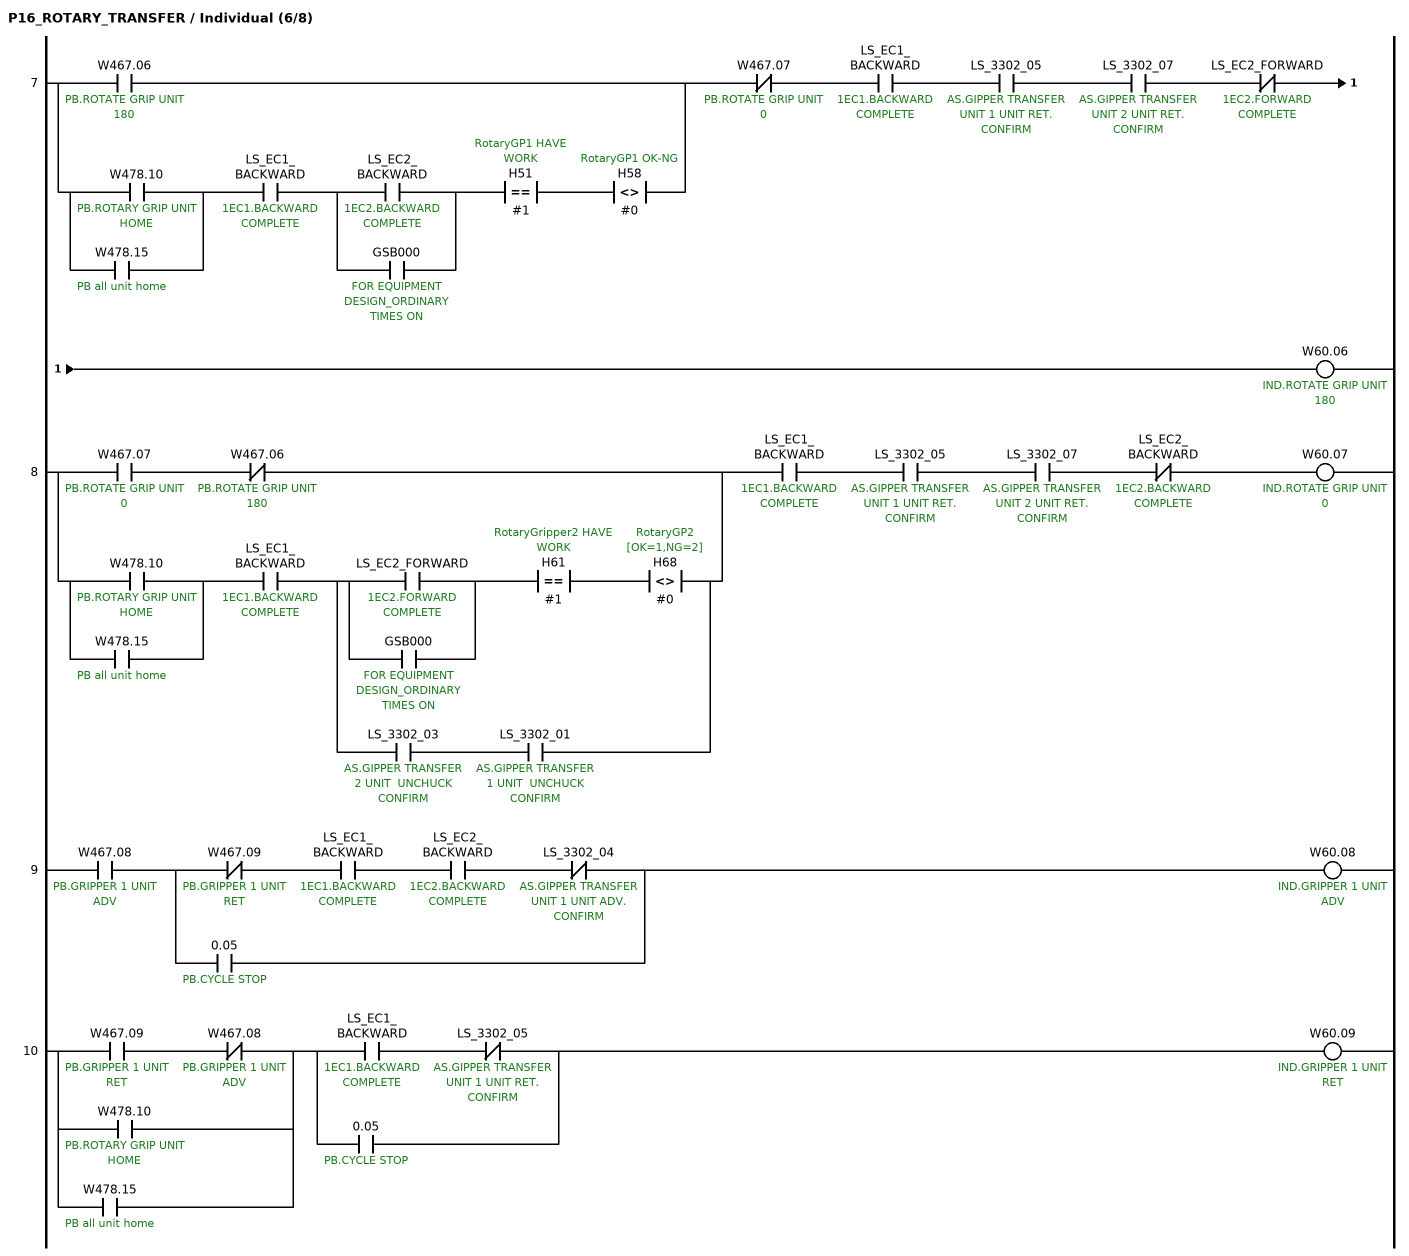
; [picture p288: P16_ROTARY_TRANSFER / Individual, rungs 7-10]
; rung 7
LD W467.06  ; PB.ROTATE GRIP UNIT 180
LD W478.10  ; PB.ROTARY GRIP UNIT HOME
OR W478.15  ; PB all unit home
AND LS_EC1_BACKWARD  ; 1EC1.BACKWARD COMPLETE
LD LS_EC2_BACKWARD  ; 1EC2.BACKWARD COMPLETE
OR GSB000  ; FOR EQUIPMENT DESIGN_ORDINARY TIMES ON
ANDLD
AND=(300) H51 #1  ; RotaryGP1 HAVE WORK
AND<>(305) H58 #0  ; RotaryGP1 OK-NG
ORLD
ANDNOT W467.07  ; PB.ROTATE GRIP UNIT 0
AND LS_EC1_BACKWARD  ; 1EC1.BACKWARD COMPLETE
AND LS_3302_05  ; AS.GIPPER TRANSFER UNIT 1 UNIT RET. CONFIRM
AND LS_3302_07  ; AS.GIPPER TRANSFER UNIT 2 UNIT RET. CONFIRM
ANDNOT LS_EC2_FORWARD  ; 1EC2.FORWARD COMPLETE
OUT W60.06  ; IND.ROTATE GRIP UNIT 180
; rung 8
LD W467.07  ; PB.ROTATE GRIP UNIT 0
ANDNOT W467.06  ; PB.ROTATE GRIP UNIT 180
LD W478.10  ; PB.ROTARY GRIP UNIT HOME
OR W478.15  ; PB all unit home
AND LS_EC1_BACKWARD  ; 1EC1.BACKWARD COMPLETE
LD LS_EC2_FORWARD  ; 1EC2.FORWARD COMPLETE
OR GSB000  ; FOR EQUIPMENT DESIGN_ORDINARY TIMES ON
AND=(300) H61 #1  ; RotaryGripper2 HAVE WORK
AND<>(305) H68 #0  ; RotaryGP2 [OK=1,NG=2]
LD LS_3302_03  ; AS.GIPPER TRANSFER 2 UNIT  UNCHUCK CONFIRM
AND LS_3302_01  ; AS.GIPPER TRANSFER 1 UNIT  UNCHUCK CONFIRM
ORLD
ANDLD
ORLD
AND LS_EC1_BACKWARD  ; 1EC1.BACKWARD COMPLETE
AND LS_3302_05  ; AS.GIPPER TRANSFER UNIT 1 UNIT RET. CONFIRM
AND LS_3302_07  ; AS.GIPPER TRANSFER UNIT 2 UNIT RET. CONFIRM
ANDNOT LS_EC2_BACKWARD  ; 1EC2.BACKWARD COMPLETE
OUT W60.07  ; IND.ROTATE GRIP UNIT 0
; rung 9
LD W467.08  ; PB.GRIPPER 1 UNIT ADV
LDNOT W467.09  ; PB.GRIPPER 1 UNIT RET
AND LS_EC1_BACKWARD  ; 1EC1.BACKWARD COMPLETE
AND LS_EC2_BACKWARD  ; 1EC2.BACKWARD COMPLETE
ANDNOT LS_3302_04  ; AS.GIPPER TRANSFER UNIT 1 UNIT ADV. CONFIRM
OR 0.05  ; PB.CYCLE STOP
ANDLD
OUT W60.08  ; IND.GRIPPER 1 UNIT ADV
; rung 10
LD W467.09  ; PB.GRIPPER 1 UNIT RET
ANDNOT W467.08  ; PB.GRIPPER 1 UNIT ADV
OR W478.10  ; PB.ROTARY GRIP UNIT HOME
OR W478.15  ; PB all unit home
LD LS_EC1_BACKWARD  ; 1EC1.BACKWARD COMPLETE
ANDNOT LS_3302_05  ; AS.GIPPER TRANSFER UNIT 1 UNIT RET. CONFIRM
OR 0.05  ; PB.CYCLE STOP
ANDLD
OUT W60.09  ; IND.GRIPPER 1 UNIT RET

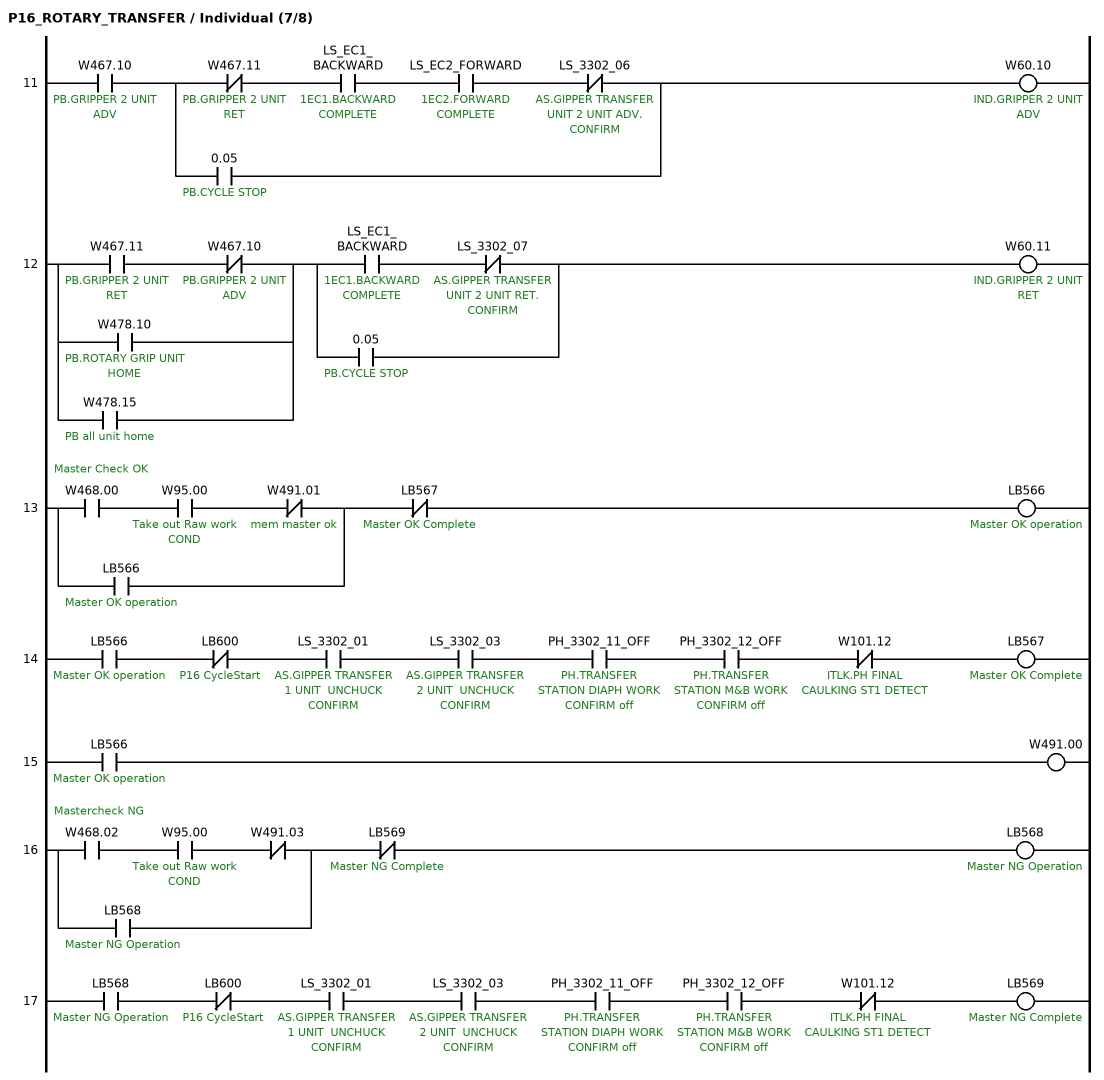
; rung 11
LD W467.10  ; PB.GRIPPER 2 UNIT ADV
LDNOT W467.11  ; PB.GRIPPER 2 UNIT RET
AND LS_EC1_BACKWARD  ; 1EC1.BACKWARD COMPLETE
AND LS_EC2_FORWARD  ; 1EC2.FORWARD COMPLETE
ANDNOT LS_3302_06  ; AS.GIPPER TRANSFER UNIT 2 UNIT ADV. CONFIRM
OR 0.05  ; PB.CYCLE STOP
ANDLD
OUT W60.10  ; IND.GRIPPER 2 UNIT ADV
; rung 12
LD W467.11  ; PB.GRIPPER 2 UNIT RET
ANDNOT W467.10  ; PB.GRIPPER 2 UNIT ADV
OR W478.10  ; PB.ROTARY GRIP UNIT HOME
OR W478.15  ; PB all unit home
LD LS_EC1_BACKWARD  ; 1EC1.BACKWARD COMPLETE
ANDNOT LS_3302_07  ; AS.GIPPER TRANSFER UNIT 2 UNIT RET. CONFIRM
OR 0.05  ; PB.CYCLE STOP
ANDLD
OUT W60.11  ; IND.GRIPPER 2 UNIT RET
; rung 13: Master Check OK
LD W468.00
AND W95.00  ; Take out Raw work COND
ANDNOT W491.01  ; mem master ok
OR LB566  ; Master OK operation
ANDNOT LB567  ; Master OK Complete
OUT LB566  ; Master OK operation
; rung 14
LD LB566  ; Master OK operation
ANDNOT LB600  ; P16 CycleStart
AND LS_3302_01  ; AS.GIPPER TRANSFER 1 UNIT  UNCHUCK CONFIRM
AND LS_3302_03  ; AS.GIPPER TRANSFER 2 UNIT  UNCHUCK CONFIRM
AND PH_3302_11_OFF  ; PH.TRANSFER STATION DIAPH WORK CONFIRM off
AND PH_3302_12_OFF  ; PH.TRANSFER STATION M&B WORK CONFIRM off
ANDNOT W101.12  ; ITLK.PH FINAL CAULKING ST1 DETECT
OUT LB567  ; Master OK Complete
; rung 15
LD LB566  ; Master OK operation
OUT W491.00
; rung 16: Mastercheck NG
LD W468.02
AND W95.00  ; Take out Raw work COND
ANDNOT W491.03
OR LB568  ; Master NG Operation
ANDNOT LB569  ; Master NG Complete
OUT LB568  ; Master NG Operation
; rung 17
LD LB568  ; Master NG Operation
ANDNOT LB600  ; P16 CycleStart
AND LS_3302_01  ; AS.GIPPER TRANSFER 1 UNIT  UNCHUCK CONFIRM
AND LS_3302_03  ; AS.GIPPER TRANSFER 2 UNIT  UNCHUCK CONFIRM
AND PH_3302_11_OFF  ; PH.TRANSFER STATION DIAPH WORK CONFIRM off
AND PH_3302_12_OFF  ; PH.TRANSFER STATION M&B WORK CONFIRM off
ANDNOT W101.12  ; ITLK.PH FINAL CAULKING ST1 DETECT
OUT LB569  ; Master NG Complete

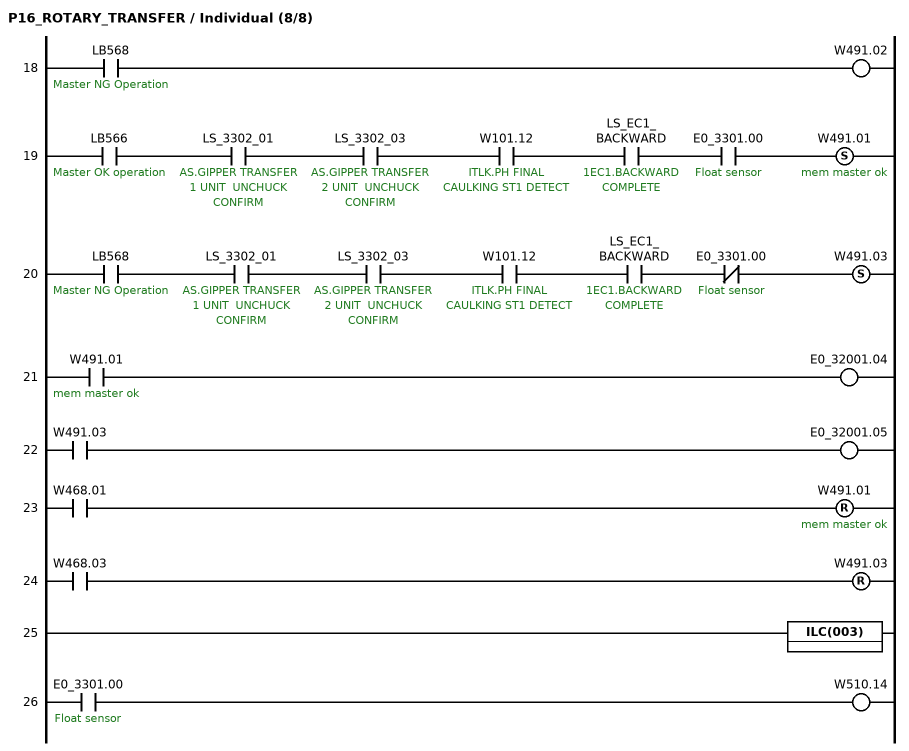
; rung 18
LD LB568  ; Master NG Operation
OUT W491.02
; rung 19
LD LB566  ; Master OK operation
AND LS_3302_01  ; AS.GIPPER TRANSFER 1 UNIT  UNCHUCK CONFIRM
AND LS_3302_03  ; AS.GIPPER TRANSFER 2 UNIT  UNCHUCK CONFIRM
AND W101.12  ; ITLK.PH FINAL CAULKING ST1 DETECT
AND LS_EC1_BACKWARD  ; 1EC1.BACKWARD COMPLETE
AND E0_3301.00  ; Float sensor
SET W491.01  ; mem master ok
; rung 20
LD LB568  ; Master NG Operation
AND LS_3302_01  ; AS.GIPPER TRANSFER 1 UNIT  UNCHUCK CONFIRM
AND LS_3302_03  ; AS.GIPPER TRANSFER 2 UNIT  UNCHUCK CONFIRM
AND W101.12  ; ITLK.PH FINAL CAULKING ST1 DETECT
AND LS_EC1_BACKWARD  ; 1EC1.BACKWARD COMPLETE
ANDNOT E0_3301.00  ; Float sensor
SET W491.03
; rung 21
LD W491.01  ; mem master ok
OUT E0_32001.04
; rung 22
LD W491.03
OUT E0_32001.05
; rung 23
LD W468.01
RSET W491.01  ; mem master ok
; rung 24
LD W468.03
RSET W491.03
; rung 25
ILC(003)
; rung 26
LD E0_3301.00  ; Float sensor
OUT W510.14

### Section END
; rung 0
END(001)

## Program P17_OK_NG_DISCHARGE (cyclic task 7)
Local symbols
LB2199 E0_46.15 BOOL  ; P16 AutoCycleEnd
LB2200 E0_41.02 BOOL  ; AUTO START BEGIN
LB2201 E0_41.03 BOOL  ; SOL.WORK FINISH TRAY DOWN
LB2202 E0_41.04 BOOL  ; SOL.WORK FINISH TRAY DOWN CONF
LB2203 E0_41.05 BOOL  ; SOL.OK PUSH UP
LB2204 E0_41.06 BOOL  ; SOL.OK PUSH UP CONF
LB2205 E0_41.07 BOOL  ; OK DISCHARGE CONFIRM
LB2206 E0_41.08 BOOL  ; SOL.OK PUSH DOWN
LB2207 E0_41.09 BOOL  ; SOL.OK PUSH DOWN CONF
LB2208 E0_41.10 BOOL  ; SOL.WORK FINISH TRAY UP
LB2209 E0_41.11 BOOL  ; SOL.WORK FINISH TRAY UP CONF
LB2210 E0_41.12 BOOL  ; AUTO START BEGIN
LB2211 E0_41.13 BOOL  ; SOL.WORK FINISH TRAY DOWN
LB2212 E0_41.14 BOOL  ; SOL.WORK FINISH TRAY DOWN CONF
LB2213 E0_41.15 BOOL  ; SOL.NG PUSH DOWN
LB2214 E0_42.00 BOOL  ; SOL.NG PUSH DOWN CONF
LB2215 E0_42.01 BOOL  ; NG DISCHARGE CONFIRM
LB2216 E0_42.02 BOOL  ; SOL.NG PUSH UP
LB2217 E0_42.03 BOOL  ; SOL.NG PUSH UP CONF
LB2218 E0_42.04 BOOL  ; SOL.WORK FINISH TRAY UP
LB2219 E0_42.05 BOOL  ; SOL.WORK FINISH TRAY UP CONF
LB2397 E0_42.06 BOOL  ; P16 OK Discharge END
LB2398 E0_42.07 BOOL  ; P16 NG Discharge END
LB2399 E0_42.08 BOOL  ; P17 AutoCycleEnd
LB432 E0_47.00 BOOL  ; IND 1 CYCLE
LB700 E0_42.09 BOOL  ; P17 CycleStart
LB701 E0_42.10 BOOL  ; P17 OK Discharge
LB702 E0_42.11 BOOL  ; P17 NG Discharge
LT2214 T3020 TIMER
LT231 T3024 TIMER
LT232 T3028 TIMER
trial_cv E0_46.02 BOOL

### Section Autorun

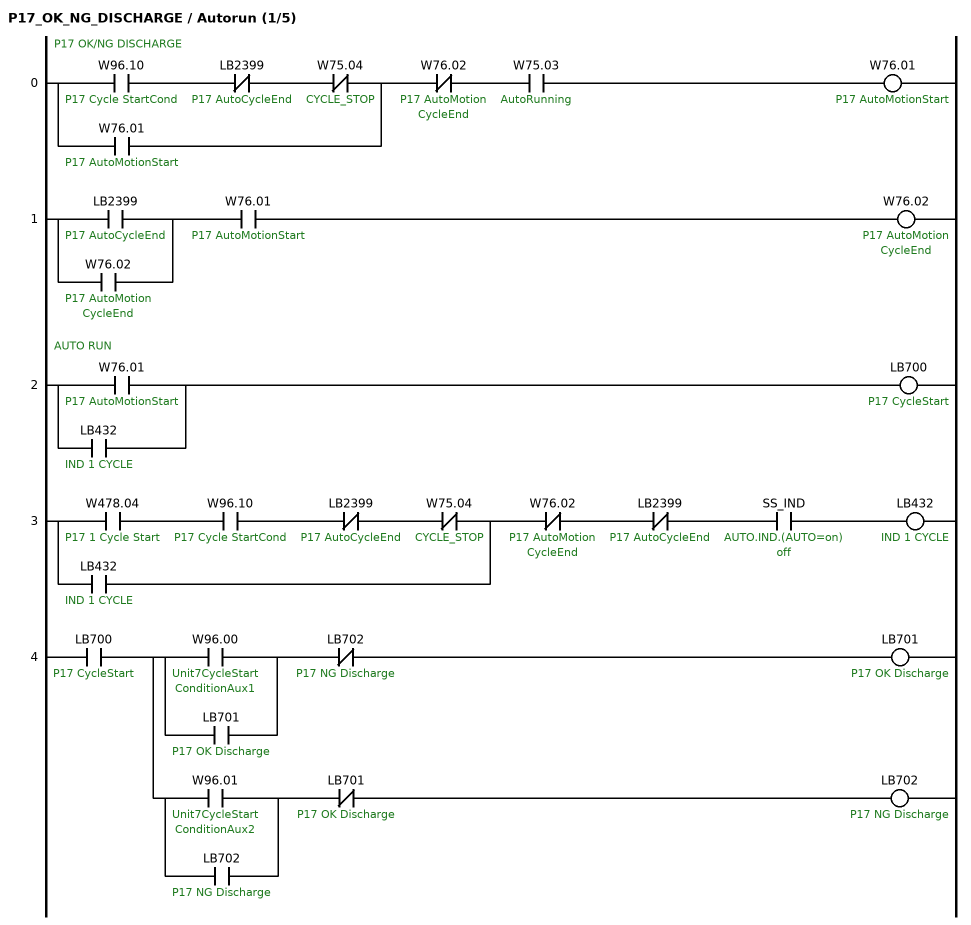
; rung 0: P17 OK/NG DISCHARGE
LD W96.10  ; P17 Cycle StartCond
ANDNOT LB2399  ; P17 AutoCycleEnd
ANDNOT W75.04  ; CYCLE_STOP
OR W76.01  ; P17 AutoMotionStart
ANDNOT W76.02  ; P17 AutoMotion CycleEnd
AND W75.03  ; AutoRunning
OUT W76.01  ; P17 AutoMotionStart
; rung 1
LD LB2399  ; P17 AutoCycleEnd
OR W76.02  ; P17 AutoMotion CycleEnd
AND W76.01  ; P17 AutoMotionStart
OUT W76.02  ; P17 AutoMotion CycleEnd
; rung 2: AUTO RUN
LD W76.01  ; P17 AutoMotionStart
OR LB432  ; IND 1 CYCLE
OUT LB700  ; P17 CycleStart
; rung 3
LD W478.04  ; P17 1 Cycle Start
AND W96.10  ; P17 Cycle StartCond
ANDNOT LB2399  ; P17 AutoCycleEnd
ANDNOT W75.04  ; CYCLE_STOP
OR LB432  ; IND 1 CYCLE
ANDNOT W76.02  ; P17 AutoMotion CycleEnd
ANDNOT LB2399  ; P17 AutoCycleEnd
AND SS_IND  ; AUTO.IND.(AUTO=on) off
OUT LB432  ; IND 1 CYCLE
; rung 4
LD LB700  ; P17 CycleStart
OUT TR0
LD W96.00  ; Unit7CycleStartConditionAux1
OR LB701  ; P17 OK Discharge
ANDLD
ANDNOT LB702  ; P17 NG Discharge
OUT LB701  ; P17 OK Discharge
LD TR0
LD W96.01  ; Unit7CycleStartConditionAux2
OR LB702  ; P17 NG Discharge
ANDLD
ANDNOT LB701  ; P17 OK Discharge
OUT LB702  ; P17 NG Discharge

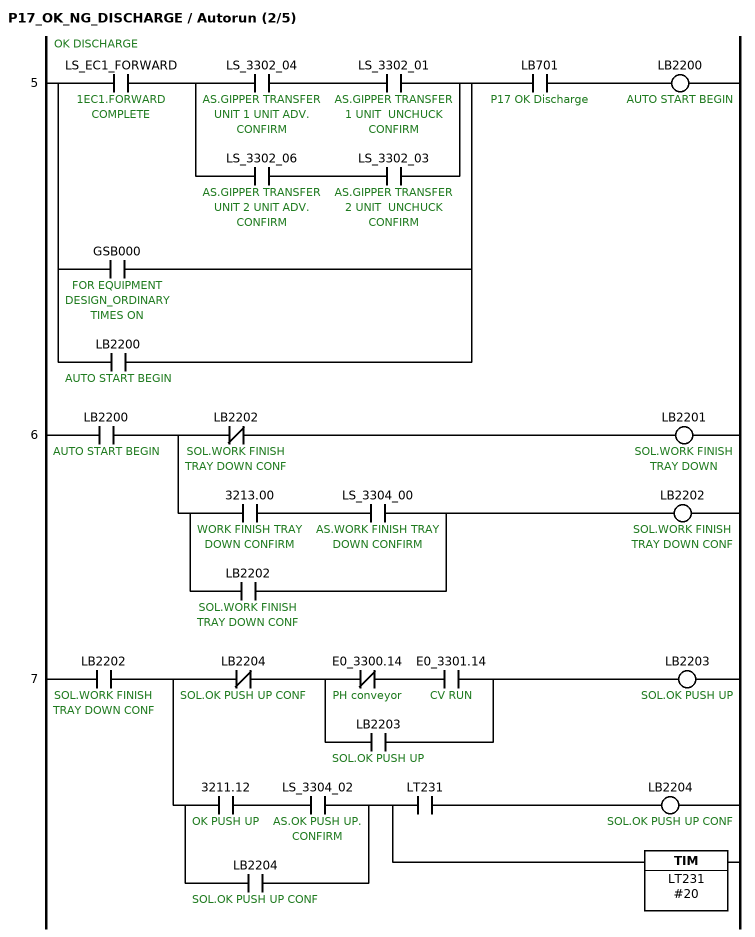
; rung 5: OK DISCHARGE
LD LS_EC1_FORWARD  ; 1EC1.FORWARD COMPLETE
LD LS_3302_04  ; AS.GIPPER TRANSFER UNIT 1 UNIT ADV. CONFIRM
AND LS_3302_01  ; AS.GIPPER TRANSFER 1 UNIT  UNCHUCK CONFIRM
LD LS_3302_06  ; AS.GIPPER TRANSFER UNIT 2 UNIT ADV. CONFIRM
AND LS_3302_03  ; AS.GIPPER TRANSFER 2 UNIT  UNCHUCK CONFIRM
ORLD
ANDLD
OR GSB000  ; FOR EQUIPMENT DESIGN_ORDINARY TIMES ON
OR LB2200  ; AUTO START BEGIN
AND LB701  ; P17 OK Discharge
OUT LB2200  ; AUTO START BEGIN
; rung 6
LD LB2200  ; AUTO START BEGIN
OUT TR0
ANDNOT LB2202  ; SOL.WORK FINISH TRAY DOWN CONF
OUT LB2201  ; SOL.WORK FINISH TRAY DOWN
LD TR0
LD 3213.00  ; WORK FINISH TRAY DOWN CONFIRM
AND LS_3304_00  ; AS.WORK FINISH TRAY DOWN CONFIRM
OR LB2202  ; SOL.WORK FINISH TRAY DOWN CONF
ANDLD
OUT LB2202  ; SOL.WORK FINISH TRAY DOWN CONF
; rung 7
LD LB2202  ; SOL.WORK FINISH TRAY DOWN CONF
OUT TR0
ANDNOT LB2204  ; SOL.OK PUSH UP CONF
LDNOT E0_3300.14  ; PH conveyor
AND E0_3301.14  ; CV RUN
OR LB2203  ; SOL.OK PUSH UP
ANDLD
OUT LB2203  ; SOL.OK PUSH UP
LD TR0
LD 3211.12  ; OK PUSH UP
AND LS_3304_02  ; AS.OK PUSH UP. CONFIRM
OR LB2204  ; SOL.OK PUSH UP CONF
ANDLD
OUT TR0
AND LT231
OUT LB2204  ; SOL.OK PUSH UP CONF
LD TR0
TIM LT231 #20

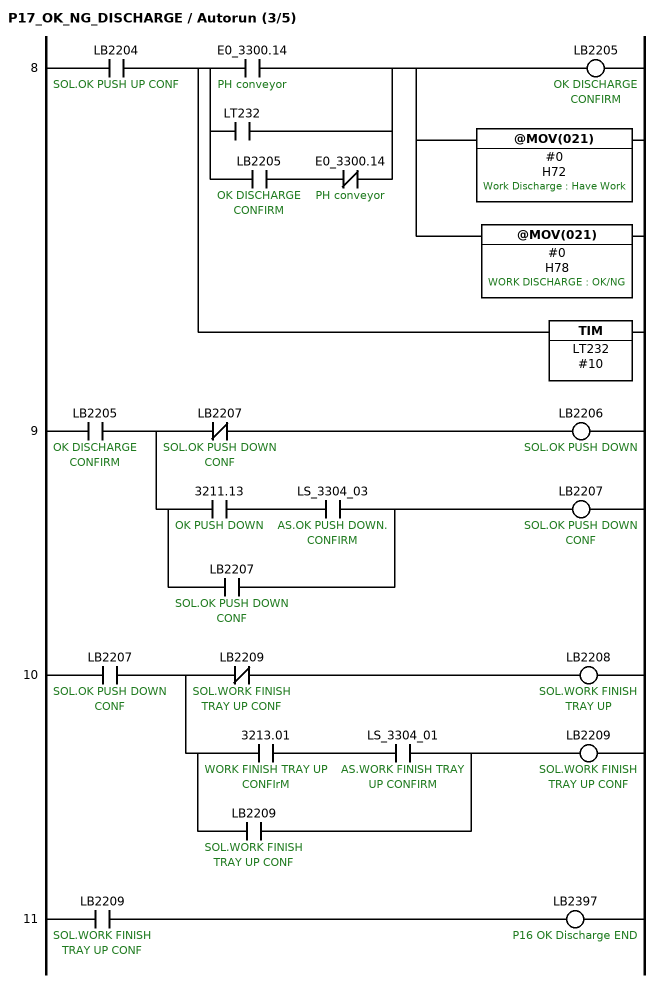
; rung 8
LD LB2204  ; SOL.OK PUSH UP CONF
OUT TR0
LD E0_3300.14  ; PH conveyor
OR LT232
LD LB2205  ; OK DISCHARGE CONFIRM
ANDNOT E0_3300.14  ; PH conveyor
ORLD
ANDLD
OUT LB2205  ; OK DISCHARGE CONFIRM
@MOV(021) #0 H72  ; Work Discharge : Have Work
@MOV(021) #0 H78  ; WORK DISCHARGE : OK/NG
LD TR0
TIM LT232 #10
; rung 9
LD LB2205  ; OK DISCHARGE CONFIRM
OUT TR0
ANDNOT LB2207  ; SOL.OK PUSH DOWN CONF
OUT LB2206  ; SOL.OK PUSH DOWN
LD TR0
LD 3211.13  ; OK PUSH DOWN
AND LS_3304_03  ; AS.OK PUSH DOWN. CONFIRM
OR LB2207  ; SOL.OK PUSH DOWN CONF
ANDLD
OUT LB2207  ; SOL.OK PUSH DOWN CONF
; rung 10
LD LB2207  ; SOL.OK PUSH DOWN CONF
OUT TR0
ANDNOT LB2209  ; SOL.WORK FINISH TRAY UP CONF
OUT LB2208  ; SOL.WORK FINISH TRAY UP
LD TR0
LD 3213.01  ; WORK FINISH TRAY UP CONFIrM
AND LS_3304_01  ; AS.WORK FINISH TRAY UP CONFIRM
OR LB2209  ; SOL.WORK FINISH TRAY UP CONF
ANDLD
OUT LB2209  ; SOL.WORK FINISH TRAY UP CONF
; rung 11
LD LB2209  ; SOL.WORK FINISH TRAY UP CONF
OUT LB2397  ; P16 OK Discharge END

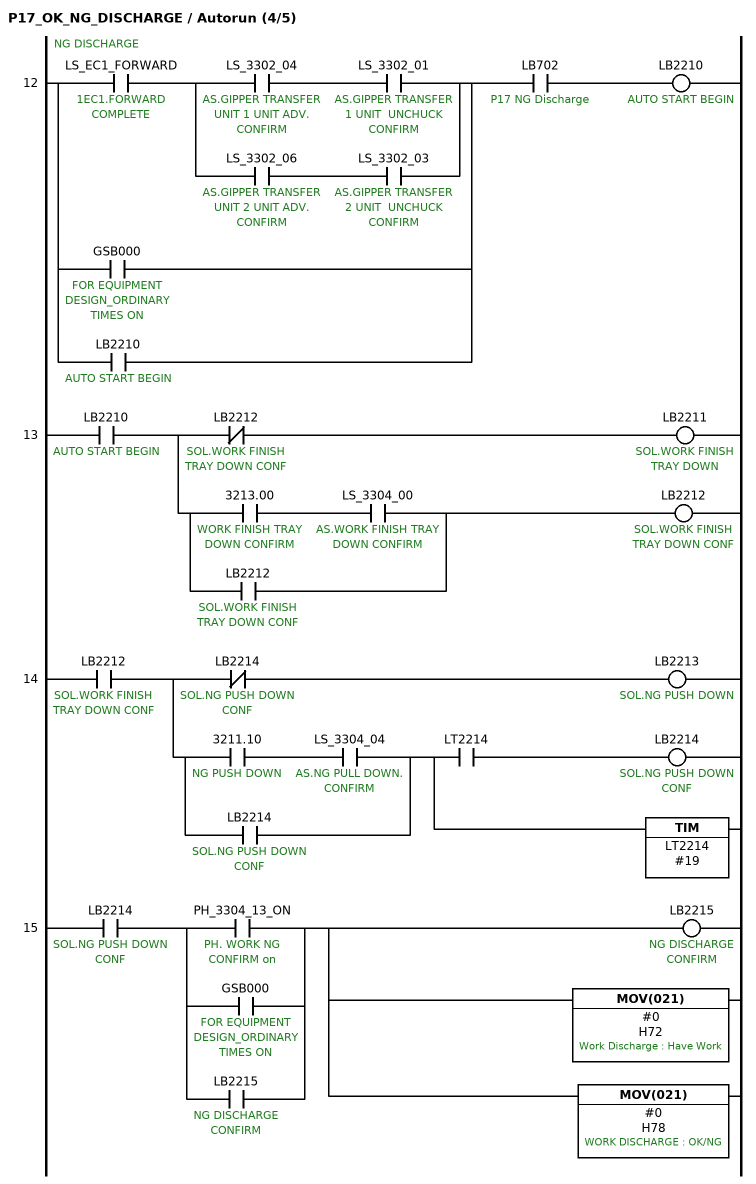
; rung 12: NG DISCHARGE
LD LS_EC1_FORWARD  ; 1EC1.FORWARD COMPLETE
LD LS_3302_04  ; AS.GIPPER TRANSFER UNIT 1 UNIT ADV. CONFIRM
AND LS_3302_01  ; AS.GIPPER TRANSFER 1 UNIT  UNCHUCK CONFIRM
LD LS_3302_06  ; AS.GIPPER TRANSFER UNIT 2 UNIT ADV. CONFIRM
AND LS_3302_03  ; AS.GIPPER TRANSFER 2 UNIT  UNCHUCK CONFIRM
ORLD
ANDLD
OR GSB000  ; FOR EQUIPMENT DESIGN_ORDINARY TIMES ON
OR LB2210  ; AUTO START BEGIN
AND LB702  ; P17 NG Discharge
OUT LB2210  ; AUTO START BEGIN
; rung 13
LD LB2210  ; AUTO START BEGIN
OUT TR0
ANDNOT LB2212  ; SOL.WORK FINISH TRAY DOWN CONF
OUT LB2211  ; SOL.WORK FINISH TRAY DOWN
LD TR0
LD 3213.00  ; WORK FINISH TRAY DOWN CONFIRM
AND LS_3304_00  ; AS.WORK FINISH TRAY DOWN CONFIRM
OR LB2212  ; SOL.WORK FINISH TRAY DOWN CONF
ANDLD
OUT LB2212  ; SOL.WORK FINISH TRAY DOWN CONF
; rung 14
LD LB2212  ; SOL.WORK FINISH TRAY DOWN CONF
OUT TR0
ANDNOT LB2214  ; SOL.NG PUSH DOWN CONF
OUT LB2213  ; SOL.NG PUSH DOWN
LD TR0
LD 3211.10  ; NG PUSH DOWN
AND LS_3304_04  ; AS.NG PULL DOWN. CONFIRM
OR LB2214  ; SOL.NG PUSH DOWN CONF
ANDLD
OUT TR0
AND LT2214
OUT LB2214  ; SOL.NG PUSH DOWN CONF
LD TR0
TIM LT2214 #19
; rung 15
LD LB2214  ; SOL.NG PUSH DOWN CONF
LD PH_3304_13_ON  ; PH. WORK NG CONFIRM on
OR GSB000  ; FOR EQUIPMENT DESIGN_ORDINARY TIMES ON
OR LB2215  ; NG DISCHARGE CONFIRM
ANDLD
OUT LB2215  ; NG DISCHARGE CONFIRM
MOV(021) #0 H72  ; Work Discharge : Have Work
MOV(021) #0 H78  ; WORK DISCHARGE : OK/NG

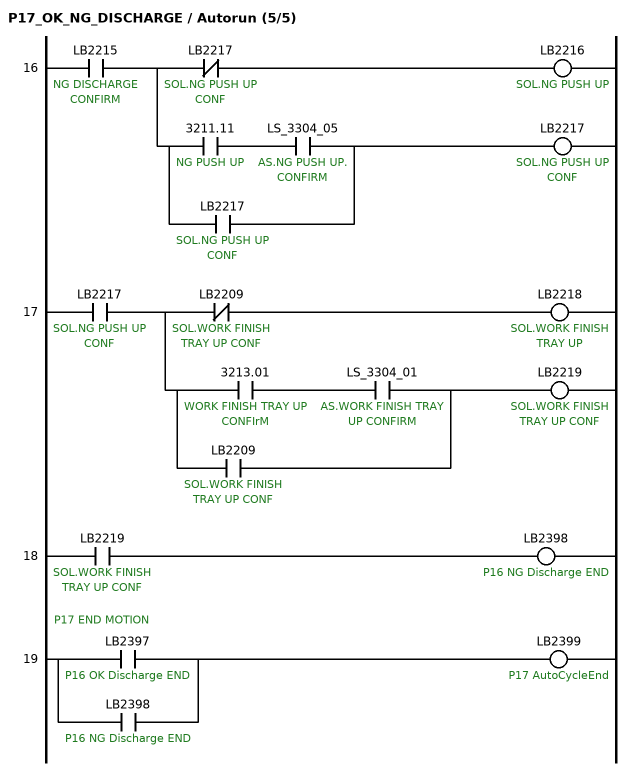
; rung 16
LD LB2215  ; NG DISCHARGE CONFIRM
OUT TR0
ANDNOT LB2217  ; SOL.NG PUSH UP CONF
OUT LB2216  ; SOL.NG PUSH UP
LD TR0
LD 3211.11  ; NG PUSH UP
AND LS_3304_05  ; AS.NG PUSH UP. CONFIRM
OR LB2217  ; SOL.NG PUSH UP CONF
ANDLD
OUT LB2217  ; SOL.NG PUSH UP CONF
; rung 17
LD LB2217  ; SOL.NG PUSH UP CONF
OUT TR0
ANDNOT LB2209  ; SOL.WORK FINISH TRAY UP CONF
OUT LB2218  ; SOL.WORK FINISH TRAY UP
LD TR0
LD 3213.01  ; WORK FINISH TRAY UP CONFIrM
AND LS_3304_01  ; AS.WORK FINISH TRAY UP CONFIRM
OR LB2209  ; SOL.WORK FINISH TRAY UP CONF
ANDLD
OUT LB2219  ; SOL.WORK FINISH TRAY UP CONF
; rung 18
LD LB2219  ; SOL.WORK FINISH TRAY UP CONF
OUT LB2398  ; P16 NG Discharge END
; rung 19: P17 END MOTION
LD LB2397  ; P16 OK Discharge END
OR LB2398  ; P16 NG Discharge END
OUT LB2399  ; P17 AutoCycleEnd

### Section Condition

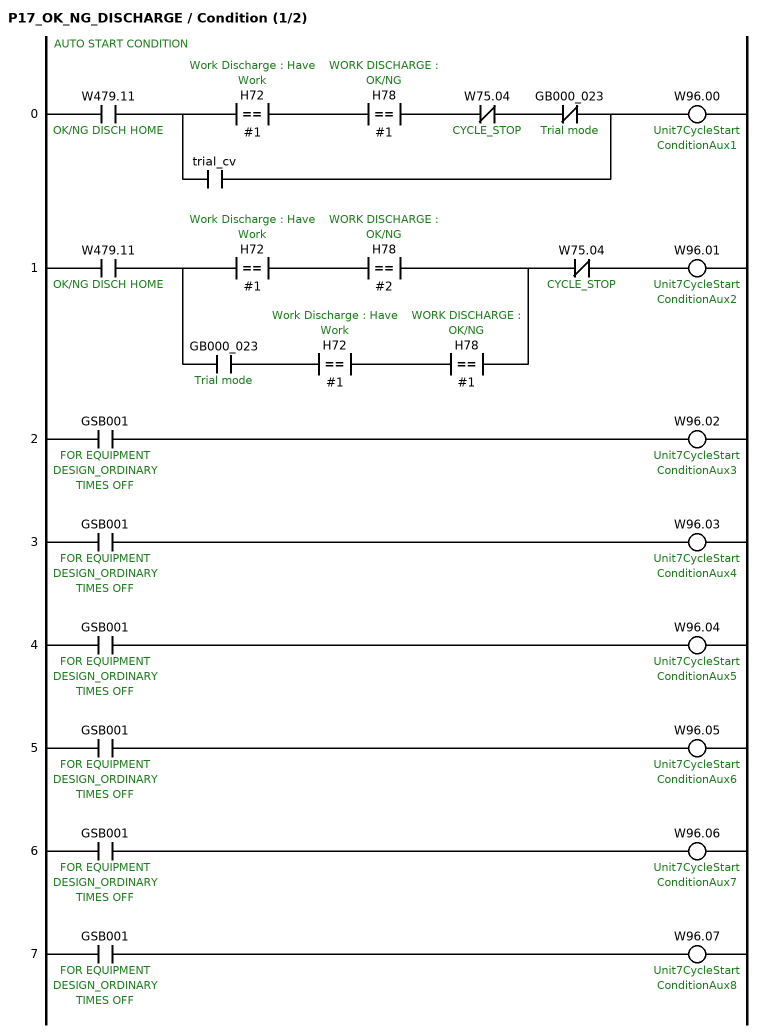
; rung 0: AUTO START CONDITION
LD W479.11  ; OK/NG DISCH HOME
LD=(300) H72 #1  ; Work Discharge : Have Work
AND=(300) H78 #1  ; WORK DISCHARGE : OK/NG
ANDNOT W75.04  ; CYCLE_STOP
ANDNOT GB000_023  ; Trial mode
OR trial_cv
ANDLD
OUT W96.00  ; Unit7CycleStartConditionAux1
; rung 1
LD W479.11  ; OK/NG DISCH HOME
LD=(300) H72 #1  ; Work Discharge : Have Work
AND=(300) H78 #2  ; WORK DISCHARGE : OK/NG
LD GB000_023  ; Trial mode
AND=(300) H72 #1  ; Work Discharge : Have Work
AND=(300) H78 #1  ; WORK DISCHARGE : OK/NG
ORLD
ANDLD
ANDNOT W75.04  ; CYCLE_STOP
OUT W96.01  ; Unit7CycleStartConditionAux2
; rung 2
LD GSB001  ; FOR EQUIPMENT DESIGN_ORDINARY TIMES OFF
OUT W96.02  ; Unit7CycleStartConditionAux3
; rung 3
LD GSB001  ; FOR EQUIPMENT DESIGN_ORDINARY TIMES OFF
OUT W96.03  ; Unit7CycleStartConditionAux4
; rung 4
LD GSB001  ; FOR EQUIPMENT DESIGN_ORDINARY TIMES OFF
OUT W96.04  ; Unit7CycleStartConditionAux5
; rung 5
LD GSB001  ; FOR EQUIPMENT DESIGN_ORDINARY TIMES OFF
OUT W96.05  ; Unit7CycleStartConditionAux6
; rung 6
LD GSB001  ; FOR EQUIPMENT DESIGN_ORDINARY TIMES OFF
OUT W96.06  ; Unit7CycleStartConditionAux7
; rung 7
LD GSB001  ; FOR EQUIPMENT DESIGN_ORDINARY TIMES OFF
OUT W96.07  ; Unit7CycleStartConditionAux8

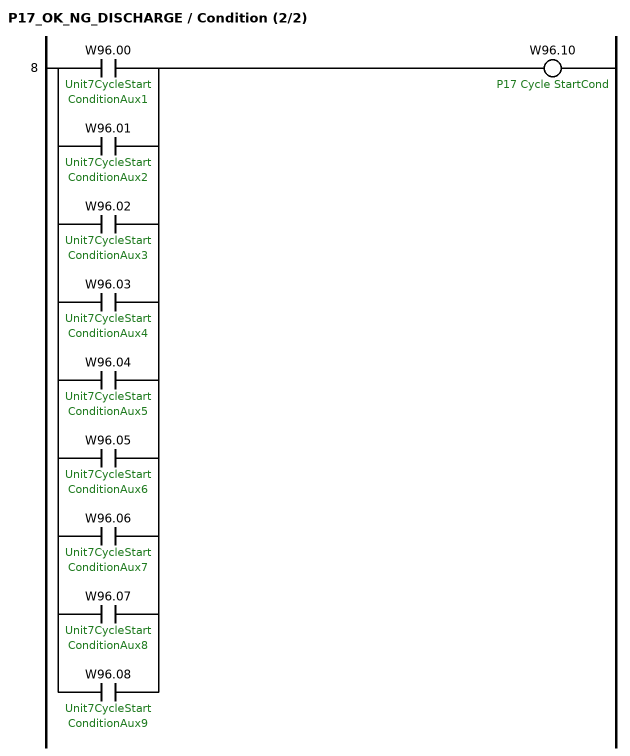
; rung 8
LD W96.00  ; Unit7CycleStartConditionAux1
OR W96.01  ; Unit7CycleStartConditionAux2
OR W96.02  ; Unit7CycleStartConditionAux3
OR W96.03  ; Unit7CycleStartConditionAux4
OR W96.04  ; Unit7CycleStartConditionAux5
OR W96.05  ; Unit7CycleStartConditionAux6
OR W96.06  ; Unit7CycleStartConditionAux7
OR W96.07  ; Unit7CycleStartConditionAux8
OR W96.08  ; Unit7CycleStartConditionAux9
OUT W96.10  ; P17 Cycle StartCond

### Section Device_Output

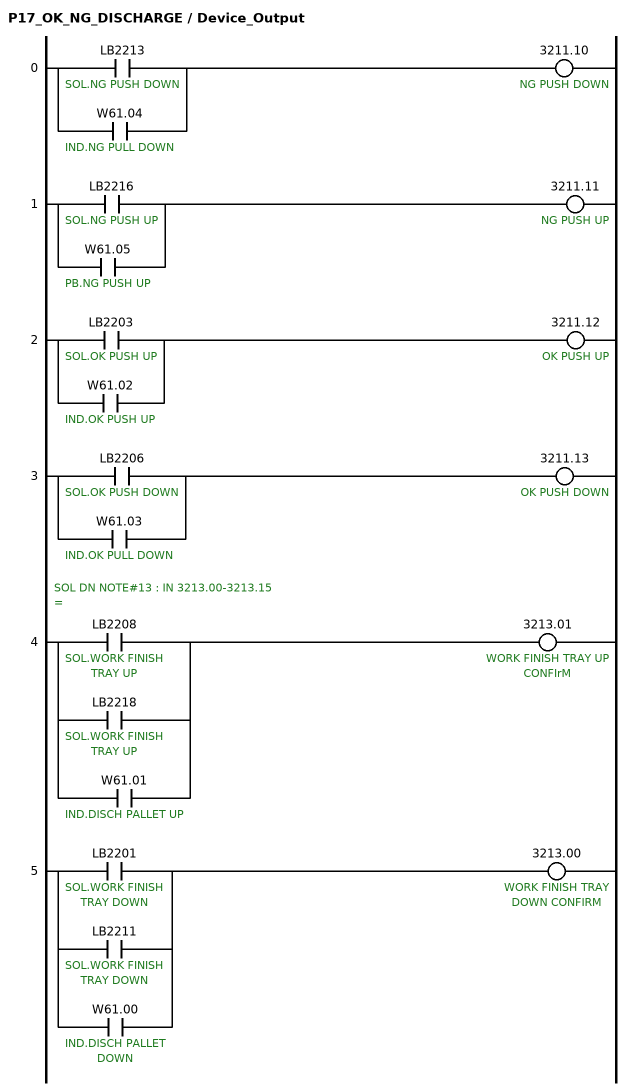
; rung 0
LD LB2213  ; SOL.NG PUSH DOWN
OR W61.04  ; IND.NG PULL DOWN
OUT 3211.10  ; NG PUSH DOWN
; rung 1
LD LB2216  ; SOL.NG PUSH UP
OR W61.05  ; PB.NG PUSH UP
OUT 3211.11  ; NG PUSH UP
; rung 2
LD LB2203  ; SOL.OK PUSH UP
OR W61.02  ; IND.OK PUSH UP
OUT 3211.12  ; OK PUSH UP
; rung 3
LD LB2206  ; SOL.OK PUSH DOWN
OR W61.03  ; IND.OK PULL DOWN
OUT 3211.13  ; OK PUSH DOWN
; rung 4: SOL DN NOTE#13 : IN 3213.00-3213.15 / =
LD LB2208  ; SOL.WORK FINISH TRAY UP
OR LB2218  ; SOL.WORK FINISH TRAY UP
OR W61.01  ; IND.DISCH PALLET UP
OUT 3213.01  ; WORK FINISH TRAY UP CONFIrM
; rung 5
LD LB2201  ; SOL.WORK FINISH TRAY DOWN
OR LB2211  ; SOL.WORK FINISH TRAY DOWN
OR W61.00  ; IND.DISCH PALLET DOWN
OUT 3213.00  ; WORK FINISH TRAY DOWN CONFIRM

### Section Station_Output

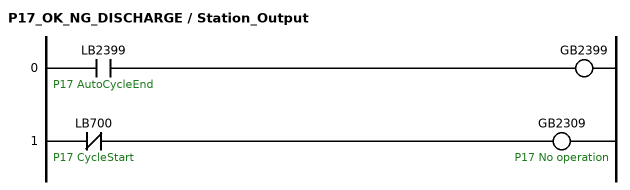
; rung 0
LD LB2399  ; P17 AutoCycleEnd
OUT GB2399
; rung 1
LDNOT LB700  ; P17 CycleStart
OUT GB2309  ; P17 No operation

### Section Individual

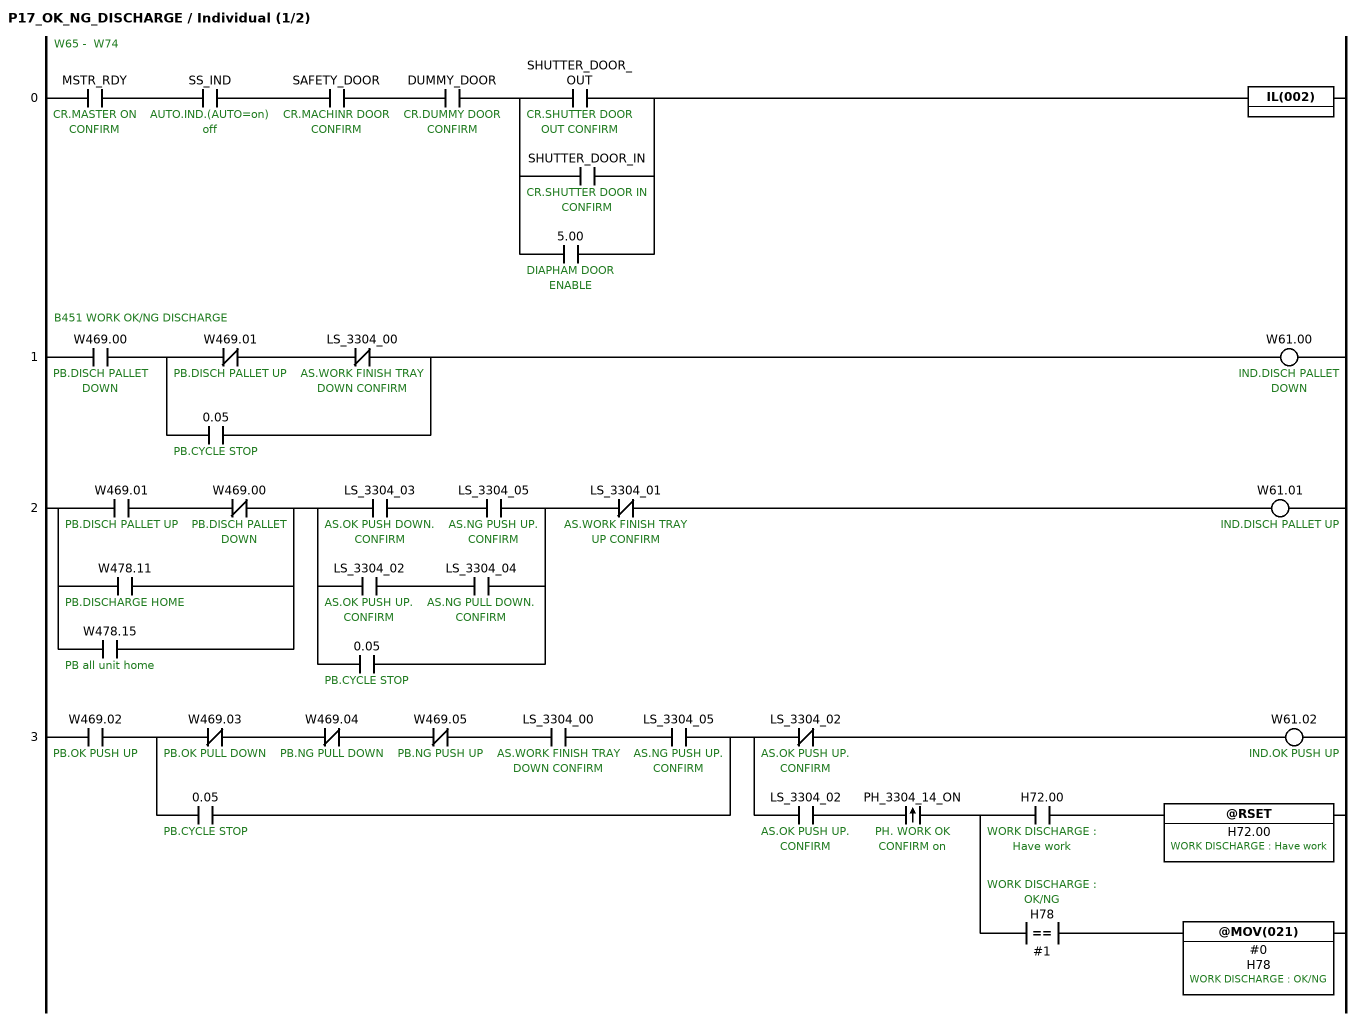
; rung 0: W65 -  W74
LD MSTR_RDY  ; CR.MASTER ON CONFIRM
AND SS_IND  ; AUTO.IND.(AUTO=on) off
AND SAFETY_DOOR  ; CR.MACHINR DOOR CONFIRM
AND DUMMY_DOOR  ; CR.DUMMY DOOR CONFIRM
LD SHUTTER_DOOR_OUT  ; CR.SHUTTER DOOR OUT CONFIRM
OR SHUTTER_DOOR_IN  ; CR.SHUTTER DOOR IN CONFIRM
OR 5.00  ; DIAPHAM DOOR ENABLE
ANDLD
IL(002)
; rung 1: B451 WORK OK/NG DISCHARGE
LD W469.00  ; PB.DISCH PALLET DOWN
LDNOT W469.01  ; PB.DISCH PALLET UP
ANDNOT LS_3304_00  ; AS.WORK FINISH TRAY DOWN CONFIRM
OR 0.05  ; PB.CYCLE STOP
ANDLD
OUT W61.00  ; IND.DISCH PALLET DOWN
; rung 2
LD W469.01  ; PB.DISCH PALLET UP
ANDNOT W469.00  ; PB.DISCH PALLET DOWN
OR W478.11  ; PB.DISCHARGE HOME
OR W478.15  ; PB all unit home
LD LS_3304_03  ; AS.OK PUSH DOWN. CONFIRM
AND LS_3304_05  ; AS.NG PUSH UP. CONFIRM
LD LS_3304_02  ; AS.OK PUSH UP. CONFIRM
AND LS_3304_04  ; AS.NG PULL DOWN. CONFIRM
ORLD
OR 0.05  ; PB.CYCLE STOP
ANDLD
ANDNOT LS_3304_01  ; AS.WORK FINISH TRAY UP CONFIRM
OUT W61.01  ; IND.DISCH PALLET UP
; rung 3
LD W469.02  ; PB.OK PUSH UP
LDNOT W469.03  ; PB.OK PULL DOWN
ANDNOT W469.04  ; PB.NG PULL DOWN
ANDNOT W469.05  ; PB.NG PUSH UP
AND LS_3304_00  ; AS.WORK FINISH TRAY DOWN CONFIRM
AND LS_3304_05  ; AS.NG PUSH UP. CONFIRM
OR 0.05  ; PB.CYCLE STOP
ANDLD
OUT TR0
ANDNOT LS_3304_02  ; AS.OK PUSH UP. CONFIRM
OUT W61.02  ; IND.OK PUSH UP
LD TR0
AND LS_3304_02  ; AS.OK PUSH UP. CONFIRM
@AND PH_3304_14_ON  ; PH. WORK OK CONFIRM on
OUT TR0
AND H72.00  ; WORK DISCHARGE : Have work
@RSET H72.00  ; WORK DISCHARGE : Have work
LD TR0
AND=(300) H78 #1  ; WORK DISCHARGE : OK/NG
@MOV(021) #0 H78  ; WORK DISCHARGE : OK/NG

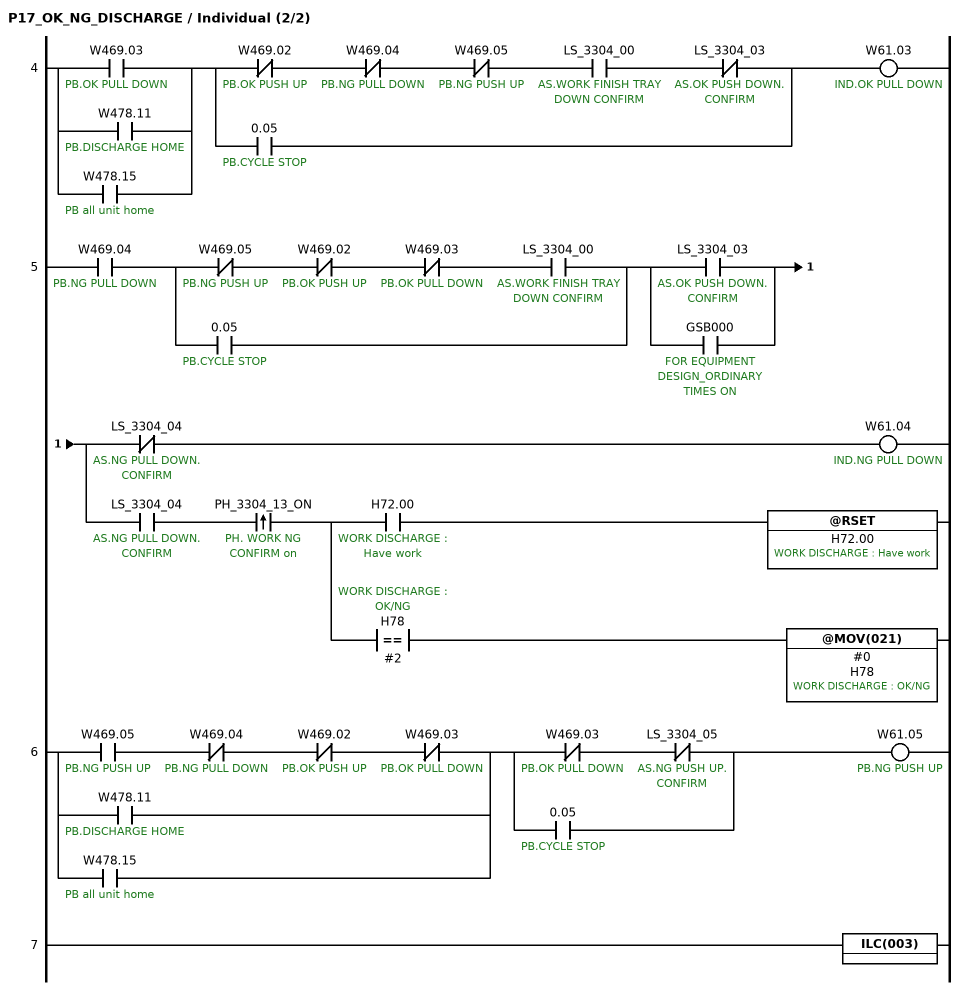
; rung 4
LD W469.03  ; PB.OK PULL DOWN
OR W478.11  ; PB.DISCHARGE HOME
OR W478.15  ; PB all unit home
LDNOT W469.02  ; PB.OK PUSH UP
ANDNOT W469.04  ; PB.NG PULL DOWN
ANDNOT W469.05  ; PB.NG PUSH UP
AND LS_3304_00  ; AS.WORK FINISH TRAY DOWN CONFIRM
ANDNOT LS_3304_03  ; AS.OK PUSH DOWN. CONFIRM
OR 0.05  ; PB.CYCLE STOP
ANDLD
OUT W61.03  ; IND.OK PULL DOWN
; rung 5
LD W469.04  ; PB.NG PULL DOWN
LDNOT W469.05  ; PB.NG PUSH UP
ANDNOT W469.02  ; PB.OK PUSH UP
ANDNOT W469.03  ; PB.OK PULL DOWN
AND LS_3304_00  ; AS.WORK FINISH TRAY DOWN CONFIRM
OR 0.05  ; PB.CYCLE STOP
ANDLD
LD LS_3304_03  ; AS.OK PUSH DOWN. CONFIRM
OR GSB000  ; FOR EQUIPMENT DESIGN_ORDINARY TIMES ON
ANDLD
OUT TR0
ANDNOT LS_3304_04  ; AS.NG PULL DOWN. CONFIRM
OUT W61.04  ; IND.NG PULL DOWN
LD TR0
AND LS_3304_04  ; AS.NG PULL DOWN. CONFIRM
@AND PH_3304_13_ON  ; PH. WORK NG CONFIRM on
OUT TR0
AND H72.00  ; WORK DISCHARGE : Have work
@RSET H72.00  ; WORK DISCHARGE : Have work
LD TR0
AND=(300) H78 #2  ; WORK DISCHARGE : OK/NG
@MOV(021) #0 H78  ; WORK DISCHARGE : OK/NG
; rung 6
LD W469.05  ; PB.NG PUSH UP
ANDNOT W469.04  ; PB.NG PULL DOWN
ANDNOT W469.02  ; PB.OK PUSH UP
ANDNOT W469.03  ; PB.OK PULL DOWN
OR W478.11  ; PB.DISCHARGE HOME
OR W478.15  ; PB all unit home
LDNOT W469.03  ; PB.OK PULL DOWN
ANDNOT LS_3304_05  ; AS.NG PUSH UP. CONFIRM
OR 0.05  ; PB.CYCLE STOP
ANDLD
OUT W61.05  ; PB.NG PUSH UP
; rung 7
ILC(003)

### Section HMI_Output

### Section END
; rung 0
END(001)